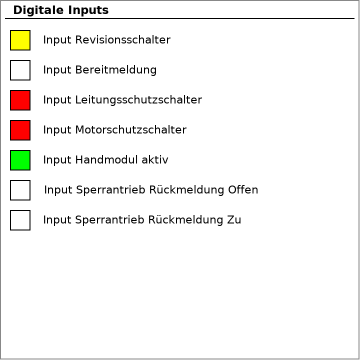
VISUALIZATION SperrAntrieb_IO0  // 360x360
VAR_INPUT
    ITF_SPERRANTRIEBIN    :   ITF_SPERRANTRIEB;	
END_VAR
    Label (40,30 320x20), "Input Revisionsschalter", invisible if: ITF_SPERRANTRIEBIN.proNotShowDI_RevisionSwitchOk
    Label (40,60 320x20), "Input Bereitmeldung", invisible if: ITF_SPERRANTRIEBIN.proNotShowDI_Ready
    Rectangle (10,30 20x20), colour toggle: ITF_SPERRANTRIEBIN.proGetDI_RevisionSwitchOK, invisible if: ITF_SPERRANTRIEBIN.proNotShowDI_RevisionSwitchOk
    Rectangle (10,60 20x20), colour toggle: ITF_SPERRANTRIEBIN.proGetDI_IsReady, invisible if: ITF_SPERRANTRIEBIN.proNotShowDI_Ready
    Rectangle (10,90 20x20), colour toggle: ITF_SPERRANTRIEBIN.proGetDI_FuseOK, invisible if: ITF_SPERRANTRIEBIN.proNotShowDI_FuseOk
    Label (40,90 320x20), "Input Leitungsschutzschalter", invisible if: ITF_SPERRANTRIEBIN.proNotShowDI_FuseOk
    Label (40,120 320x20), "Input Motorschutzschalter", invisible if: ITF_SPERRANTRIEBIN.proNotShowDI_ActuatorFuseOk
    Rectangle (10,120 20x20), colour toggle: ITF_SPERRANTRIEBIN.proGetDI_ActuatorFuseOk, invisible if: ITF_SPERRANTRIEBIN.proNotShowDI_ActuatorFuseOk
    Label (40,150 320x20), "Input Handmodul aktiv", invisible if: ITF_SPERRANTRIEBIN.proNotShowDI_ActuatorHand
    Rectangle (10,150 20x20), colour toggle: ITF_SPERRANTRIEBIN.proGetDI_ActuatorHand, invisible if: ITF_SPERRANTRIEBIN.proNotShowDI_ActuatorHand
    Label (10,0 350x20), "Digitale Inputs"
    Rectangle (10,210 20x20), colour toggle: ITF_SPERRANTRIEBIN.proGetDI_RükIsClosed, invisible if: ITF_SPERRANTRIEBIN.proNotShowDI_RükIsOpen
    Label (40,210 320x20), "Input Sperrantrieb Rückmeldung Zu", invisible if: ITF_SPERRANTRIEBIN.proNotShowDI_RükIsOpen
    Rectangle (10,180 20x20), colour toggle: ITF_SPERRANTRIEBIN.proGetDI_RükIsOpen, invisible if: ITF_SPERRANTRIEBIN.proNotShowDI_RükIsOpen
    Label (41,180 320x20), "Input Sperrantrieb Rückmeldung Offen", invisible if: ITF_SPERRANTRIEBIN.proNotShowDI_RükIsOpen
    Line (5,18) (354,18)
END_VISUALIZATION

// 40 Visualizations/POPUP/IO/SperrAntrieb_IO
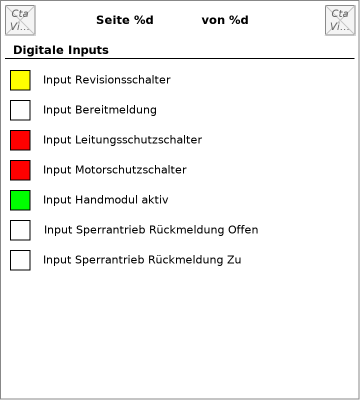
VISUALIZATION SperrAntrieb_IO  // 360x400
VAR_INPUT
    ITF_SPERRANTRIEBIN    :   ITF_SPERRANTRIEB;	
END_VAR
VAR
    uiPage  :   UINT;
    uiMin   :   UINT    := 0;
    uiMax   :   UINT    := 1;
END_VAR
    Frame (0,40 360x360), frame switch variable: uiPage
        shows SperrAntrieb_IO0(ITF_SPERRANTRIEBIN := ITF_SPERRANTRIEBIN)
        shows SperrAntrieb_IO1(ITF_SPERRANTRIEBIN := ITF_SPERRANTRIEBIN)
        shows AT_ParameterIO2(ITF_Parameter := ITF_Parameter)
        shows AT_ParameterIO3(ITF_Parameter := ITF_Parameter)
    Image (325,5 30x30), invisible if: uiPage = uiMax, image: CtaVisSymbols.ImagePool.arrow-right_square
        OnMouseClick: execute {
            uiPage := uiPage + 1;
            IF uiPage >= uiMax THEN
                uiPage := uiMax;
            END_IF;
        }
    Image (5,5 30x30), invisible if: uiPage = uiMin, image: CtaVisSymbols.ImagePool.arrow-left_square
        OnMouseClick: execute {
            uiPage := uiPage - 1;
            IF uiPage <= uiMin THEN
                uiPage := uiMin;
            END_IF;
        }
    Textfield (175,5 100x30), "von %d", text variable: uiMax
    Textfield (75,5 100x30), "Seite %d", text variable: uiPage
END_VISUALIZATION

// 40 Visualizations/POPUP/IO/SperrAntrieb_IO1
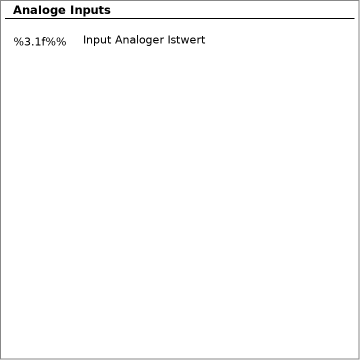
VISUALIZATION SperrAntrieb_IO1  // 360x360
VAR_INPUT
    ITF_SPERRANTRIEBIN    :   ITF_SPERRANTRIEB;	
END_VAR
    Label (80,30 280x20), "Input Analoger Istwert", invisible if: ITF_SPERRANTRIEBIN.proNotShowAI_ActualPosition
    Label (10,0 350x20), "Analoge Inputs"
    Textfield (10,32 60x20), "%3.1f%%", text variable: ITF_SPERRANTRIEBIN.proGetAI_ActualPosition, invisible if: ITF_SPERRANTRIEBIN.proNotShowAI_ActualPosition
    Line (5,18) (354,18)
END_VISUALIZATION

// 40 Visualizations/ICON/SperrAntrieb_BASE/Ventile/Klappe/Motor_Right/MR_Klappe_ZU
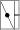
VISUALIZATION MR_Klappe_ZU  // 20x30
    Polygon (0,0) (14,30) (14,0)
    Polygon (0,0) (0,30) (14,30)
    Ellipse (5,13 4x4)
    Line (20,15) (14,15)
END_VISUALIZATION

// 40 Visualizations/ICON/SperrAntrieb_BASE/Ventile/Klappe/Motor_Left/ML_Klappe_ZU
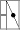
VISUALIZATION ML_Klappe_ZU  // 20x30
    Polygon (6,0) (20,30) (20,0)
    Polygon (6,0) (6,30) (20,30)
    Ellipse (11,13 4x4)
    Line (6,15) (0,15)
END_VISUALIZATION

// 40 Visualizations/ICON/SperrAntrieb_BASE/Ventile/Klappe/Motor_Above/MA_Klappe_ZU
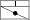
VISUALIZATION MA_Klappe_ZU  // 30x20
    Polygon (0,6) (30,20) (30,6)
    Polygon (0,6) (0,20) (30,20)
    Ellipse (13,11 4x4)
    Line (15,0) (15,6)
END_VISUALIZATION

// 40 Visualizations/ICON/SperrAntrieb_BASE/Ventile/Klappe/Motor_Below/MB_Klappe_ZU
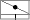
VISUALIZATION MB_Klappe_ZU  // 30x20
    Polygon (0,0) (30,14) (30,0)
    Polygon (0,0) (0,14) (30,14)
    Ellipse (13,5 4x4)
    Line (15,14) (15,20)
END_VISUALIZATION

// 40 Visualizations/ICON/SperrAntrieb_BASE/Icons/Motor_Left/Icon_ML_Klappe
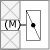
VISUALIZATION Icon_ML_Klappe  // 50x50
VAR_INPUT
    ITF_SPERRANTRIEB_IN   :   ITF_SPERRANTRIEB;	
END_VAR
    Frame (5,17 15x15)
        shows Motor(ITF_SPERRANTRIEB_IN := ITF_SPERRANTRIEB_IN)
    Frame (20,10 20x30), invisible if: ITF_SPERRANTRIEB_IN.proGetDI_RükIsClosed OR( ITF_SPERRANTRIEB_IN.proKlappenStatus = 2) OR( ITF_SPERRANTRIEB_IN.proKlappenStatus =3)
        shows ML_Klappe_AUF()
    Frame (20,10 20x30), invisible if: ITF_SPERRANTRIEB_IN.proGetDI_RükIsOpen OR (ITF_SPERRANTRIEB_IN.proKlappenStatus = 4) OR (ITF_SPERRANTRIEB_IN.proKlappenStatus = 1)
        shows ML_Klappe_ZU()
    Image (0,0 20x20), invisible if: NOT ITF_SPERRANTRIEB_IN.proIsWarning, image: CtaVisSymbols.ImagePool.CtaWarning
    Image (0,30 20x20), invisible if: NOT ITF_SPERRANTRIEB_IN.proIsHandOnOrOff, image: CtaVisSymbols.ImagePool.front_hand_Yellow
    Image (0,30 20x20), invisible if: NOT ITF_SPERRANTRIEB_IN.proHandOff, image: CtaVisSymbols.ImagePool.front_hand_Yellow_Off
END_VISUALIZATION

// 40 Visualizations/ICON/SperrAntrieb_BASE/Icons/Motor_Right/Icon_MR_Klappe
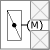
VISUALIZATION Icon_MR_Klappe  // 50x50
VAR_INPUT
    ITF_SPERRANTRIEB_IN   :   ITF_SPERRANTRIEB;	
END_VAR
    Frame (27,18 15x15)
        shows Motor(ITF_SPERRANTRIEB_IN := ITF_SPERRANTRIEB_IN)
    Frame (7,10 20x30), invisible if: ITF_SPERRANTRIEB_IN.proGetDI_RükIsClosed OR( ITF_SPERRANTRIEB_IN.proKlappenStatus = 2) OR( ITF_SPERRANTRIEB_IN.proKlappenStatus =3)
        shows MR_Klappe_AUF()
    Frame (7,10 20x30), invisible if: ITF_SPERRANTRIEB_IN.proGetDI_RükIsOpen OR (ITF_SPERRANTRIEB_IN.proKlappenStatus = 4) OR (ITF_SPERRANTRIEB_IN.proKlappenStatus = 1)
        shows MR_Klappe_ZU()
    Image (30,0 20x20), invisible if: NOT ITF_SPERRANTRIEB_IN.proIsWarning, image: CtaVisSymbols.ImagePool.CtaWarning
    Image (30,30 20x20), invisible if: NOT ITF_SPERRANTRIEB_IN.proIsHandOnOrOff, image: CtaVisSymbols.ImagePool.front_hand_Yellow
    Image (30,30 20x20), invisible if: NOT ITF_SPERRANTRIEB_IN.proHandOff, image: CtaVisSymbols.ImagePool.front_hand_Yellow_Off
END_VISUALIZATION

// 40 Visualizations/ICON/SperrAntrieb_BASE/Icons/Motor_Above/Icon_MA_Klappe
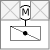
VISUALIZATION Icon_MA_Klappe  // 50x50
VAR_INPUT
    ITF_SPERRANTRIEB_IN   :   ITF_SPERRANTRIEB;	
END_VAR
    Frame (18,5 15x15)
        shows Motor(ITF_SPERRANTRIEB_IN := ITF_SPERRANTRIEB_IN)
    Frame (10,20 30x20), invisible if: ITF_SPERRANTRIEB_IN.proGetDI_RükIsClosed OR( ITF_SPERRANTRIEB_IN.proKlappenStatus = 2) OR( ITF_SPERRANTRIEB_IN.proKlappenStatus =3)
        shows MA_Klappe_AUF()
    Frame (10,20 30x20), invisible if: ITF_SPERRANTRIEB_IN.proGetDI_RükIsOpen OR (ITF_SPERRANTRIEB_IN.proKlappenStatus = 4) OR (ITF_SPERRANTRIEB_IN.proKlappenStatus = 1)
        shows MA_Klappe_ZU()
    Image (0,0 20x20), invisible if: NOT ITF_SPERRANTRIEB_IN.proIsWarning, image: CtaVisSymbols.ImagePool.CtaWarning
    Image (30,0 20x20), invisible if: NOT ITF_SPERRANTRIEB_IN.proIsHandOnOrOff, image: CtaVisSymbols.ImagePool.front_hand_Yellow
    Image (30,0 20x20), invisible if: NOT ITF_SPERRANTRIEB_IN.proHandOff, image: CtaVisSymbols.ImagePool.front_hand_Yellow_Off
END_VISUALIZATION

// 40 Visualizations/ICON/SperrAntrieb_BASE/Icons/Motor_Below/Icon_MB_Klappe
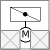
VISUALIZATION Icon_MB_Klappe  // 50x50
VAR_INPUT
    ITF_SPERRANTRIEB_IN   :   ITF_SPERRANTRIEB;	
END_VAR
    Frame (18,27 15x15)
        shows Motor(ITF_SPERRANTRIEB_IN := ITF_SPERRANTRIEB_IN)
    Frame (10,7 30x20), invisible if: ITF_SPERRANTRIEB_IN.proGetDI_RükIsClosed OR( ITF_SPERRANTRIEB_IN.proKlappenStatus = 2) OR( ITF_SPERRANTRIEB_IN.proKlappenStatus =3)
        shows MB_Klappe_AUF()
    Frame (10,7 30x22), invisible if: ITF_SPERRANTRIEB_IN.proGetDI_RükIsOpen OR (ITF_SPERRANTRIEB_IN.proKlappenStatus = 4) OR (ITF_SPERRANTRIEB_IN.proKlappenStatus = 1)
        shows MB_Klappe_ZU()
    Image (0,30 20x20), invisible if: NOT ITF_SPERRANTRIEB_IN.proIsWarning, image: CtaVisSymbols.ImagePool.CtaWarning
    Image (30,30 20x20), invisible if: NOT ITF_SPERRANTRIEB_IN.proIsHandOnOrOff, image: CtaVisSymbols.ImagePool.front_hand_Yellow
    Image (30,30 20x20), invisible if: NOT ITF_SPERRANTRIEB_IN.proHandOff, image: CtaVisSymbols.ImagePool.front_hand_Yellow_Off
END_VISUALIZATION

// 40 Visualizations/ICON/SperrAntrieb_BASE/Ventile/Klappe/Motor_Above/MA_Klappe_AUF
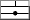
VISUALIZATION MA_Klappe_AUF  // 30x20
    Rectangle (0,6 30x14)
    Line (15,0) (15,6)
    Line (0,13) (30,13)
    Ellipse (13,11 4x4)
END_VISUALIZATION

// 40 Visualizations/ICON/SperrAntrieb_LEFT/Motor_Above/SperrAntrieb_MA_Flap_LA_CheckQuerry
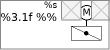
VISUALIZATION SperrAntrieb_MA_Flap_LA_CheckQuerry  // 110x50
VAR_INPUT
    ITF_SPERRANTRIEB_IN   :   ITF_SPERRANTRIEB;
    stExklParameter		:   STRING[40];	
END_VAR
    Frame (0,0 110x50)
        shows SperrAntrieb_MA_Flap_LA_CheckEnabled(ITF_SPERRANTRIEB_IN := ITF_SPERRANTRIEB_IN, stExklParameter := stExklParameter)
END_VISUALIZATION

// 40 Visualizations/ICON/SperrAntrieb_LEFT/Motor_Above/SperrAntrieb_MA_Flap_Txt_L_Above
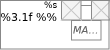
VISUALIZATION SperrAntrieb_MA_Flap_Txt_L_Above  // 110x50
VAR_INPUT
    ITF_SPERRANTRIEB_IN		:   ITF_SPERRANTRIEB;	
END_VAR
VAR_INPUT CONSTANT
    stExklParameter		:   STRING[40] := ' ';	
END_VAR
VAR CONSTANT
	uiIconNr				:	UINT := 0;
END_VAR
    Frame (0,0 110x50), invisible if: NOT fcCheckQuerryReturnIcon(_ITF_In := ITF_SPERRANTRIEB_IN,_uiIconNr_In := uiIconNr)
        shows SperrAntrieb_MA_Flap_LA_CheckQuerry(ITF_SPERRANTRIEB_IN := ITF_SPERRANTRIEB_IN, stExklParameter := stExklParameter)
        shows S_AT_MA_Flap_LA_CheckQuerry()
END_VISUALIZATION

// 40 Visualizations/ICON/SperrAntrieb_RIGHT/Motor_Above/SperrAntrieb_MA_Flap_RA_CheckEnabled
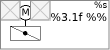
VISUALIZATION SperrAntrieb_MA_Flap_RA_CheckEnabled  // 110x50
VAR_INPUT
    ITF_SPERRANTRIEB_IN   :   ITF_SPERRANTRIEB;
    stExklParameter		:   STRING[40];	
END_VAR
    Frame (0,0 50x50), invisible if: NOT ITF_SPERRANTRIEB_IN.proIsEnabled
        shows Icon_MA_Klappe(ITF_SPERRANTRIEB_IN := ITF_SPERRANTRIEB_IN)
    Frame (50,0 60x25), invisible if: NOT ITF_SPERRANTRIEB_IN.proIsEnabled
        shows ValueUpDwn(ITF_SPERRANTRIEB_IN := ITF_SPERRANTRIEB_IN, uiTextAusrichtung := 4)
    Rectangle (0,0 110x50)
        OnMouseClick:  Dialog=SperrAntrieb_POPUP, Parameters={stExklParameter: stExklParameter, ITF_SPERRANTRIEBIN: ITF_SPERRANTRIEB_IN, uiPopUpGruppe: 0}, OpenCentered=True
END_VISUALIZATION

// 40 Visualizations/ICON/SperrAntrieb_RIGHT/Motor_Above/SperrAntrieb_MA_Flap_RA_CheckQuerry
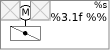
VISUALIZATION SperrAntrieb_MA_Flap_RA_CheckQuerry  // 110x50
VAR_INPUT
    ITF_SPERRANTRIEB_IN   :   ITF_SPERRANTRIEB;
    stExklParameter		:   STRING[40];	
END_VAR
    Frame (0,0 110x50)
        shows SperrAntrieb_MA_Flap_RA_CheckEnabled(ITF_SPERRANTRIEB_IN := ITF_SPERRANTRIEB_IN, stExklParameter := stExklParameter)
END_VISUALIZATION

// 40 Visualizations/ICON/SperrAntrieb_RIGHT/Motor_Above/SperrAntrieb_MA_Flap_Txt_R_Above
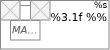
VISUALIZATION SperrAntrieb_MA_Flap_Txt_R_Above  // 110x50
VAR_INPUT
    ITF_SPERRANTRIEB_IN		:   ITF_SPERRANTRIEB;	
END_VAR
VAR_INPUT CONSTANT
    stExklParameter		:   STRING[40] := ' ';	
END_VAR
VAR CONSTANT
	uiIconNr				:	UINT := 4;
END_VAR
    Frame (0,0 110x50), invisible if: NOT fcCheckQuerryReturnIcon(_ITF_In := ITF_SPERRANTRIEB_IN,_uiIconNr_In := uiIconNr)
        shows SperrAntrieb_MA_Flap_RA_CheckQuerry(ITF_SPERRANTRIEB_IN := ITF_SPERRANTRIEB_IN, stExklParameter := stExklParameter)
        shows Icon()
END_VISUALIZATION

// 40 Visualizations/ICON/SperrAntrieb_LEFT/Motor_Above/SperrAntrieb_MA_Flap_LA_CheckEnabled
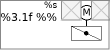
VISUALIZATION SperrAntrieb_MA_Flap_LA_CheckEnabled  // 110x50
VAR_INPUT
    ITF_SPERRANTRIEB_IN   :   ITF_SPERRANTRIEB;
    stExklParameter		:   STRING[40];	
END_VAR
    Frame (61,0 50x50), invisible if: NOT ITF_SPERRANTRIEB_IN.proIsEnabled
        shows Icon_MA_Klappe(ITF_SPERRANTRIEB_IN := ITF_SPERRANTRIEB_IN)
    Frame (0,0 60x25), invisible if: NOT ITF_SPERRANTRIEB_IN.proIsEnabled
        shows ValueUpDwn(ITF_SPERRANTRIEB_IN := ITF_SPERRANTRIEB_IN, uiTextAusrichtung := 6)
    Rectangle (0,0 110x50)
        OnMouseClick:  Dialog=SperrAntrieb_POPUP, Parameters={stExklParameter: stExklParameter, ITF_SPERRANTRIEBIN: ITF_SPERRANTRIEB_IN, uiPopUpGruppe: 0}, OpenCentered=True
END_VISUALIZATION

// 40 Visualizations/ICON/SperrAntrieb_RIGHT/Motor_Below/SperrAntrieb_MB_Flap_RB_CheckEnabled
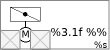
VISUALIZATION SperrAntrieb_MB_Flap_RB_CheckEnabled  // 110x50
VAR_INPUT
    ITF_SPERRANTRIEB_IN   :   ITF_SPERRANTRIEB;
    stExklParameter		:   STRING[40];	
END_VAR
    Frame (0,0 50x50), invisible if: NOT ITF_SPERRANTRIEB_IN.proIsEnabled
        shows Icon_MB_Klappe(ITF_SPERRANTRIEB_IN := ITF_SPERRANTRIEB_IN)
    Frame (50,25 60x25), invisible if: NOT ITF_SPERRANTRIEB_IN.proIsEnabled
        shows ValueDwnUp(ITF_SPERRANTRIEB_IN := ITF_SPERRANTRIEB_IN, uiTextAusrichtung := 4)
    Rectangle (0,0 110x50)
        OnMouseClick:  Dialog=SperrAntrieb_POPUP, Parameters={stExklParameter: stExklParameter, ITF_SPERRANTRIEBIN: ITF_SPERRANTRIEB_IN, uiPopUpGruppe: 0}, OpenCentered=True
END_VISUALIZATION

// 40 Visualizations/ICON/SperrAntrieb_RIGHT/Motor_Below/SperrAntrieb_MB_Flap_RB_CheckQuerry
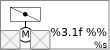
VISUALIZATION SperrAntrieb_MB_Flap_RB_CheckQuerry  // 110x50
VAR_INPUT
    ITF_SPERRANTRIEB_IN   :   ITF_SPERRANTRIEB;
    stExklParameter		:   STRING[40];	
END_VAR
    Frame (0,0 110x50)
        shows SperrAntrieb_MB_Flap_RB_CheckEnabled(ITF_SPERRANTRIEB_IN := ITF_SPERRANTRIEB_IN, stExklParameter := stExklParameter)
END_VISUALIZATION

// 40 Visualizations/ICON/SperrAntrieb_RIGHT/Motor_Below/SperrAntrieb_MB_Flap_Right_Txt_R_Below
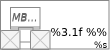
VISUALIZATION SperrAntrieb_MB_Flap_Right_Txt_R_Below  // 110x50
VAR_INPUT
    ITF_SPERRANTRIEB_IN		:   ITF_SPERRANTRIEB;	
END_VAR
VAR_INPUT CONSTANT
    stExklParameter		:   STRING[40] := ' ';	
END_VAR
VAR CONSTANT
	uiIconNr				:	UINT := 5;
END_VAR
    Frame (0,0 110x50), invisible if: NOT fcCheckQuerryReturnIcon(_ITF_In := ITF_SPERRANTRIEB_IN,_uiIconNr_In := uiIconNr)
        shows SperrAntrieb_MB_Flap_RB_CheckQuerry(ITF_SPERRANTRIEB_IN := ITF_SPERRANTRIEB_IN, stExklParameter := stExklParameter)
        shows Icon()
END_VISUALIZATION

// 40 Visualizations/ICON/SperrAntrieb_RIGHT/Motor_Right/Above/SperrAntrieb_MR_Flap_Txt_R_Above
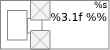
VISUALIZATION SperrAntrieb_MR_Flap_Txt_R_Above  // 110x50
VAR_INPUT
    ITF_SPERRANTRIEB_IN		:   ITF_SPERRANTRIEB;	
END_VAR
VAR_INPUT CONSTANT
    stExklParameter		:   STRING[40] := ' ';	
END_VAR
VAR CONSTANT
	uiIconNr				:	UINT := 6;
END_VAR
    Frame (0,0 110x50), invisible if: NOT fcCheckQuerryReturnIcon(_ITF_In := ITF_SPERRANTRIEB_IN,_uiIconNr_In := uiIconNr)
        shows SperrAntrieb_MR_Flap_RA_CheckQuerry(ITF_SPERRANTRIEB_IN := ITF_SPERRANTRIEB_IN, stExklParameter := stExklParameter)
        shows Icon()
END_VISUALIZATION

// 40 Visualizations/ICON/SperrAntrieb_RIGHT/Motor_Right/Above/SperrAntrieb_MR_Flap_RA_CheckQuerry
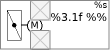
VISUALIZATION SperrAntrieb_MR_Flap_RA_CheckQuerry  // 110x50
VAR_INPUT
    ITF_SPERRANTRIEB_IN   :   ITF_SPERRANTRIEB;
    stExklParameter		:   STRING[40];	
END_VAR
    Frame (0,0 110x50)
        shows SperrAntrieb_MR_Flap_RA_CheckEnabled(ITF_SPERRANTRIEB_IN := ITF_SPERRANTRIEB_IN, stExklParameter := stExklParameter)
END_VISUALIZATION

// 40 Visualizations/ICON/SperrAntrieb_RIGHT/Motor_Right/Above/SperrAntrieb_MR_Flap_RA_CheckEnabled
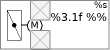
VISUALIZATION SperrAntrieb_MR_Flap_RA_CheckEnabled  // 110x50
VAR_INPUT
    ITF_SPERRANTRIEB_IN   :   ITF_SPERRANTRIEB;
    stExklParameter		:   STRING[40];	
END_VAR
    Frame (0,0 50x50), invisible if: NOT ITF_SPERRANTRIEB_IN.proIsEnabled
        shows Icon_MR_Klappe(ITF_SPERRANTRIEB_IN := ITF_SPERRANTRIEB_IN)
    Frame (50,0 60x25), invisible if: NOT ITF_SPERRANTRIEB_IN.proIsEnabled
        shows ValueUpDwn(ITF_SPERRANTRIEB_IN := ITF_SPERRANTRIEB_IN, uiTextAusrichtung := 4)
    Rectangle (0,0 110x50)
        OnMouseClick:  Dialog=SperrAntrieb_POPUP, Parameters={stExklParameter: stExklParameter, ITF_SPERRANTRIEBIN: ITF_SPERRANTRIEB_IN, uiPopUpGruppe: 0}, OpenCentered=True
END_VISUALIZATION

// 40 Visualizations/ICON/SperrAntrieb_RIGHT/Motor_Right/Below/SperrAntrieb_MR_Flap_Txt_R_Below
